FUNCTION F_CoolTank : BOOL
VAR_INPUT
	rTank : REFERENCE TO ST_Tank;
END_VAR
VAR
	fCoolingSpeed : REAL := 3;
	fRequiredTemperature : REAL := 50;
END_VAR

IF __ISVALIDREF(rTank) THEN
	IF rTank.fTemperature > fRequiredTemperature THEN
		rTank.fTemperature := rTank.fTemperature - fCoolingSpeed;
	ELSE
		rTank.bAlarm := FALSE;
		rTank.fTemperature := rTank.fTemperature + fCoolingSpeed;
	END_IF
END_IF

END_FUNCTION

(* stored: Version 1.1.0.1, ProductVersion 3.1.4024.16
   POU F_CoolTank: Id {6b86b570-fb14-4991-ae3f-71ce75cc8823}, SpecialFunc None *)
